INTERFACE I_Dimmable EXTENDS __SYSTEM.IQueryInterface

METHOD M_SetControlLevel
VAR_INPUT
	nControlLevel	:	BYTE;
END_VAR
END_METHOD

METHOD M_RecallMinLevel
VAR_INPUT
END_VAR
END_METHOD

PROPERTY nMaxLevel : BYTE
GET
END_GET
SET
END_SET
END_PROPERTY

PROPERTY nControlLevel : BYTE
SET
END_SET
GET
END_GET
END_PROPERTY

PROPERTY nMinLevel : BYTE
SET
END_SET
GET
END_GET
END_PROPERTY

END_INTERFACE

(* stored: Version 1.1.0.1, ProductVersion 3.1.0.20
   Itf I_Dimmable: Id {b7492116-7ecc-429f-aca2-bf88e4725b00}
   Method M_SetControlLevel: Id {193a878d-92d6-4792-b65a-bdf92939c23d}
   Method M_RecallMinLevel: Id {36b8e14a-3d46-4770-9bea-53d6acf4f89b}
   Property nMaxLevel: Id {9ba1e131-5917-46f3-a92a-e210574144ca}
   Get Get: Id {6181fca1-d4cb-450d-a673-988326c63c34}
   Set Set: Id {cf8de8b8-4e5f-45d2-9fb5-6ef5ca5764ae}
   Property nControlLevel: Id {9eb81d6f-aa2c-479d-80eb-70339adc4290}
   Set Set: Id {45f91477-79b3-4ccf-9b3c-d632b1a7d2b6}
   Get Get: Id {c1148527-b01d-40b3-821c-500dac438454}
   Property nMinLevel: Id {b8b863f9-435f-4235-ac3c-dbabdc47862c}
   Set Set: Id {38bb7413-3274-4835-93dd-5065c3bf1e3a}
   Get Get: Id {4d2c8918-f47d-4e28-a1a1-0ab8e4d5376e} *)
